TEXTLIST ManualPageTitle
  10001 = '==Line1=OP0010'
  10005 = 'Page 5 s1'
  10004 = 'Page 4 s1'
  10003 = 'Page 3 s1'
  10002 = 'Page 2 s1'
  10006 = 'Page 6 s1'
  20001 = 'Page 1 s2'
  20002 = 'Page 2 s2'
  20003 = 'Page 3 s2'
  20004 = 'Page 4 s2'
  20005 = 'Page 5 s2'
  20006 = 'Page 6 s2'
  30001 = 'Page 1 s3'
  30002 = 'Page 2 s3'
  30003 = 'Page 3 s3'
  30004 = 'Page 4 s3'
  30005 = 'Page 5 s3'
  30006 = 'Page 6 s3'
  40001 = 'Page 1 s4'
  40002 = 'Page 2 s4'
  40003 = 'Page 3 s4'
  40004 = 'Page 4 s4'
  40005 = 'Page 5 s4'
  40006 = 'Page 6 s4'
  50001 = 'Page 1 s5'
  50002 = 'Page 2 s5'
  50003 = 'Page 3 s5'
  50004 = 'Page 4 s5'
  50005 = 'Page 5 s5'
  50006 = 'Page 6 s5'
  60001 = 'Page 1 s6'
  60002 = 'Page 2 s6'
  60003 = 'Page 3 s6'
  60004 = 'Page 4 s6'
  60005 = 'Page 5 s6'
  60006 = 'Page 6 s6'
   = ''
END_TEXTLIST

(* stored: Version 1.1.0.1, ProductVersion 3.1.4024.12
   TextList ManualPageTitle: Id {1a499272-26b1-4d40-80b4-0f1248606b35} *)
